TYPE ST_TagData :
STRUCT
	fBlinkIndex			: LREAL;	// An ever increasing number (32-bit integer) that gets incremented every time the tag blinks.
	staCustomSensors	: ARRAY[0..GVL_PozyxParameters.cnMaxCustomSensors] OF ST_CustomSensor;
END_STRUCT
END_TYPE

(* stored: Version 1.1.0.1, ProductVersion 3.1.4024.3
   DUT ST_TagData: Id {0f847e2a-5546-414b-a261-5e3dab58beca} *)
